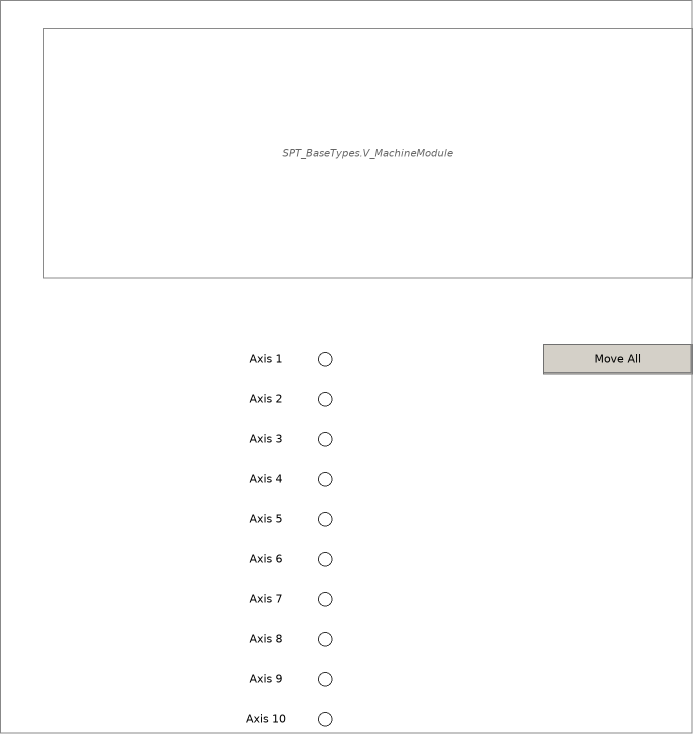
VISUALIZATION Visualization  // 693x734
    Frame (43,28 650x250)
        shows SPT_BaseTypes.V_MachineModule(HMI := MAIN.Machine.PackMLBaseModule_HMI)
    RadioButton (316,344 150x30), variable: MAIN.Machine.AxisAssignment[1]
        Areas[0]: Text=Left
        Areas[1]: Text=Right
    Label (226,344 80x30), "Axis 1"
    RadioButton (316,384 150x30), variable: MAIN.Machine.AxisAssignment[2]
        Areas[0]: Text=Left
        Areas[1]: Text=Right
    Label (226,384 80x30), "Axis 2"
    RadioButton (316,424 150x30), variable: MAIN.Machine.AxisAssignment[3]
        Areas[0]: Text=Left
        Areas[1]: Text=Right
    Label (226,424 80x30), "Axis 3"
    RadioButton (316,464 150x30), variable: MAIN.Machine.AxisAssignment[4]
        Areas[0]: Text=Left
        Areas[1]: Text=Right
    Label (226,464 80x30), "Axis 4"
    RadioButton (316,504 150x30), variable: MAIN.Machine.AxisAssignment[5]
        Areas[0]: Text=Left
        Areas[1]: Text=Right
    Label (226,504 80x30), "Axis 5"
    RadioButton (316,544 150x30), variable: MAIN.Machine.AxisAssignment[6]
        Areas[0]: Text=Left
        Areas[1]: Text=Right
    Label (226,544 80x30), "Axis 6"
    RadioButton (316,584 150x30), variable: MAIN.Machine.AxisAssignment[7]
        Areas[0]: Text=Left
        Areas[1]: Text=Right
    Label (226,584 80x30), "Axis 7"
    RadioButton (316,624 150x30), variable: MAIN.Machine.AxisAssignment[8]
        Areas[0]: Text=Left
        Areas[1]: Text=Right
    Label (226,624 80x30), "Axis 8"
    RadioButton (316,664 150x30), variable: MAIN.Machine.AxisAssignment[9]
        Areas[0]: Text=Left
        Areas[1]: Text=Right
    Label (226,664 80x30), "Axis 9"
    RadioButton (316,704 150x30), variable: MAIN.Machine.AxisAssignment[10]
        Areas[0]: Text=Left
        Areas[1]: Text=Right
    Label (226,704 80x30), "Axis 10"
    Button (543,344 150x30), "Move All"
        tap MAIN.Machine.HMI.Cmd.MoveAll
END_VISUALIZATION

(* stored: Version 1.1.0.1
   Visu Visualization: Id {865fa0fc-20ce-46e4-9410-7017db8f6b03} *)
